# B&R Automation Studio project RobotNewEra (part 14)

#### HmiEditorLocal.typ - Local data types
```iecst
(********************************************************************
 * COPYRIGHT --
 ********************************************************************
 * Program: HmiEdit
 * File: HmiEdit.typ
 * Author: renj
 * Created: October 21, 2014
 ********************************************************************
 * Local data types of program HmiEdit
 ********************************************************************)

TYPE
	HmiEditorInternalStateType :
		(
		HMIEDITOR_WAIT,
		HMIEDITOR_READ,
		HMIEDITOR_LOADED,
		HMIEDITOR_WRITE_WAIT,
		HMIEDITOR_ERROR
		);
	HmiEditorInternalType : 	STRUCT
		State : HmiEditorInternalStateType;
	END_STRUCT;
END_TYPE
```

#### HmiEditorLocal.var - Local variables
```iecst
(********************************************************************
 * COPYRIGHT --
 ********************************************************************
 * Program: HmiEdit
 * File: HmiEdit.var
 * Author: renj
 * Created: October 21, 2014
 ********************************************************************
 * Local variables of program HmiEdit
 ********************************************************************)
VAR
	Internal : HmiEditorInternalType := (0);
	pSystem : REFERENCE TO System_Type;
	pCnc : REFERENCE TO Cnc_Type;
	pAxes : REFERENCE TO ARRAY[0..MAX_AX_MINUS_ONE] OF Axes_Type;
END_VAR
```

### Program Logical/HmiHandling/HmiEditor/HmiFileVar (IEC) - File Read Write

#### HmiFileCtrlVar.st - Implementation code
```iecst
(********************************************************************
 * COPYRIGHT --
 ********************************************************************
 * Program: HmiFile
 * File: HmiFileCtrlVar.st
 * Author: renj
 * Created: October 29, 2014
 ********************************************************************
 * Implementation of program HmiFile
 ********************************************************************)

PROGRAM _INIT

END_PROGRAM

PROGRAM _CYCLIC

	CASE Internal.State OF

		HMIFILE_IDLE:

			HmiFileCtrlVar.Output.Status.Busy := FALSE;

			IF HmiFileCtrlVar.Input.Command.Read THEN

				Internal.State := HMIFILE_OPEN;
				HmiFileCtrlVar.Output.Status.ReadOK := FALSE;
				HmiFileCtrlVar.Output.Status.Busy := TRUE;

			END_IF

			IF HmiFileCtrlVar.Input.Command.Write THEN

				Internal.State := HMIFILE_DELETE;
				HmiFileCtrlVar.Output.Status.WriteOK := FALSE;
				HmiFileCtrlVar.Output.Status.Busy := TRUE;
			END_IF

		HMIFILE_OPEN:

			FileOpen_0.enable	:= TRUE;
			FileOpen_0.pDevice 	:= ADR(HmiFileCtrlVar.Input.Parameter.FileDevice);
			FileOpen_0.pFile 	:= ADR(HmiFileCtrlVar.Input.Parameter.FileName);
			FileOpen_0.mode 	:= fiREAD_WRITE;
			(* FB Call *)
			FileOpen_0();

			(* Get FBK output information *)
			Internal.FileIdent := FileOpen_0.ident;
			wStatus := FileOpen_0.status;

			IF (wStatus = 0) THEN

				Internal.State := HMIFILE_READ;

			ELSIF (wStatus <> 65535) THEN
				(* Verify status (20708 -> File doesn't exist) *)
				IF (wStatus = 20708) THEN

				END_IF

				IF (wStatus = 20799) THEN
					wError := FileIoGetSysError();
				END_IF

				IF HmiFileCtrlVar.Input.Command.Read THEN

					HmiFileCtrlVar.Input.Command.Read := FALSE;

				ELSIF HmiFileCtrlVar.Input.Command.Write THEN

					HmiFileCtrlVar.Input.Command.Write := FALSE;

				END_IF

				Internal.State := HMIFILE_ERROR;

			END_IF

		HMIFILE_READ:

			(**** Read data from file ****)
			(* Initialize file read structure *)
			FileReadEx_0.enable		:= TRUE;
			FileReadEx_0.ident     	:= Internal.FileIdent;
			FileReadEx_0.pDest     	:= HmiFileCtrlVar.Input.Parameter.StringBufferAdr;
			FileReadEx_0.len	   	:= HmiFileCtrlVar.Input.Parameter.StringBufferSize;

			(* Call FBK *)
			FileReadEx_0();
			(* Get status *)
			wStatus := FileReadEx_0.status;
			(* Verify status *)
			IF wStatus = 0 THEN

				Internal.FileByte := FileReadEx_0.bytesread;

				Internal.State := HMIFILE_CLOSE;

			ELSIF (wStatus <> 65535) THEN

				IF (wStatus = 20799) THEN
					wError := FileIoGetSysError();
				END_IF

				IF HmiFileCtrlVar.Input.Command.Read THEN

					HmiFileCtrlVar.Input.Command.Read := FALSE;

				ELSIF HmiFileCtrlVar.Input.Command.Write THEN

					HmiFileCtrlVar.Input.Command.Write := FALSE;

				END_IF

				Internal.State := HMIFILE_ERROR;

			END_IF

		HMIFILE_DELETE:
			(* Initialize file delete structure *)
			FileDelete_0.enable  := 1;
			FileDelete_0.pDevice := ADR(HmiFileCtrlVar.Input.Parameter.FileDevice);
			FileDelete_0.pName   :=ADR(HmiFileCtrlVar.Input.Parameter.FileName);
			(* Call FBK *)
			FileDelete_0();
			(* Get status *)
			wStatus := FileDelete_0.status;

			(* Verify status *)
			IF wStatus = 0 THEN
				Internal.State := HMIFILE_CREATE;
			ELSIF (wStatus <> 65535) THEN

				IF (wStatus = 20799) THEN
					wError := FileIoGetSysError();
				END_IF

				IF HmiFileCtrlVar.Input.Command.Write THEN

					HmiFileCtrlVar.Input.Command.Write := FALSE;

				END_IF

				Internal.State := HMIFILE_ERROR;

			END_IF

		HMIFILE_CREATE:
			(* Initialize file create structure *)
			FileCreate_0.enable  := 1;
			FileCreate_0.pDevice := ADR(HmiFileCtrlVar.Input.Parameter.FileDevice);
			FileCreate_0.pFile   := ADR(HmiFileCtrlVar.Input.Parameter.FileName);
			(* Call FBK *)
			FileCreate_0();
			(* Get FBK output information *)
			Internal.FileIdent := FileCreate_0.ident;
			wStatus := FileCreate_0.status;
			(* Verify status *)
			IF wStatus = 0 THEN
				Internal.State := HMIFILE_WRITE;
			ELSIF (wStatus <> 65535) THEN

				IF (wStatus = 20799) THEN
					wError := FileIoGetSysError();
				END_IF

				IF HmiFileCtrlVar.Input.Command.Write THEN

					HmiFileCtrlVar.Input.Command.Write := FALSE;

				END_IF

				Internal.State := HMIFILE_ERROR;

			END_IF

		HMIFILE_WRITE:
			(**** WRITE File ****)
			(* Initialize file close structure *)
			FileWriteEx_0.enable	:= TRUE;
			FileWriteEx_0.ident		:= Internal.FileIdent;

			FileWriteEx_0.len		:= HmiFileCtrlVar.Input.Parameter.StringBufferSize;
			FileWriteEx_0.pSrc		:= HmiFileCtrlVar.Input.Parameter.StringBufferAdr;;

			(* Call FBK *)
			FileWriteEx_0();

			(* Get status *)
			wStatus := FileWriteEx_0.status;

			(* Verify status *)
			IF wStatus = 0 THEN
				Internal.State := HMIFILE_CLOSE;
			ELSIF (wStatus <> 65535) THEN

				IF (wStatus = 20799) THEN
					wError := FileIoGetSysError();
				END_IF

				IF HmiFileCtrlVar.Input.Command.Read THEN

					HmiFileCtrlVar.Input.Command.Read := FALSE;

				ELSIF HmiFileCtrlVar.Input.Command.Write THEN

					HmiFileCtrlVar.Input.Command.Write := FALSE;

				END_IF

				Internal.State := HMIFILE_ERROR;

			END_IF

		HMIFILE_CLOSE:
			(**** Close file ****)
			(* Initialize file close structure *)
			FileClose_0.enable	:= TRUE;
			FileClose_0.ident	:= Internal.FileIdent;

			(* Call FBK *)
			FileClose_0();

			(* Get status *)
			wStatus := FileClose_0.status;

			IF wStatus = 0 THEN

				IF HmiFileCtrlVar.Input.Command.Read THEN

					HmiFileCtrlVar.Output.Status.ReadOK := TRUE;

					HmiFileCtrlVar.Input.Command.Read := FALSE;

				ELSIF HmiFileCtrlVar.Input.Command.Write THEN

					HmiFileCtrlVar.Output.Status.WriteOK := TRUE;

					HmiFileCtrlVar.Input.Command.Write := FALSE;

				END_IF

				Internal.State := HMIFILE_IDLE;

			ELSIF (wStatus <> 65535) THEN

				IF (wStatus = 20799) THEN
					wError := FileIoGetSysError();
				END_IF

				IF HmiFileCtrlVar.Input.Command.Read THEN

					HmiFileCtrlVar.Input.Command.Read := FALSE;

				ELSIF HmiFileCtrlVar.Input.Command.Write THEN

					HmiFileCtrlVar.Input.Command.Write := FALSE;

				END_IF

				Internal.State := HMIFILE_ERROR;

			END_IF

		HMIFILE_ERROR:

			IF HmiFileCtrlVar.Input.Command.AckError THEN

				HmiFileCtrlVar.Input.Command.AckError := 0;
				Internal.State := HMIFILE_IDLE;

			END_IF

	END_CASE

END_PROGRAM
```

#### HmiFileVarLocal.var - Local variables
```iecst
(********************************************************************
 * COPYRIGHT --
 ********************************************************************
 * Program: HmiFile
 * File: HmiFileLocal.var
 * Author: renj
 * Created: October 29, 2014
 ********************************************************************
 * Local variables of program HmiFile
 ********************************************************************)
VAR
	FileOpen_0 : FileOpen := (0);
	FileClose_0 : FileClose := (0);
	FileReadEx_0 : FileReadEx := (0);
	FileDelete_0 : FileDelete := (0);
	FileCreate_0 : FileCreate := (0);
	FileWriteEx_0 : FileWriteEx := (0);
	wStatus : UINT := 0;
	wError : UINT := 0;
	Internal : HmiFileCtrlInternal_Type := (0);
END_VAR
```

### Package Logical/HmiHandling/HmiAlarm - Alarm Page

### Program Logical/HmiHandling/HmiAlarm/HmiAlarm (IEC) - Alarm Ctrl Page

#### HmiAlarm.st - Implementation code
```iecst
(********************************************************************
 * COPYRIGHT --
 ********************************************************************
 * Program: HmiAlarm
 * File: HmiAlarm.st
 * Author: renj
 * Created: October 14, 2014
 ********************************************************************
 * Implementation of program HmiAlarm
 ********************************************************************)

PROGRAM _INIT

END_PROGRAM

PROGRAM _CYCLIC

	IF HmiGlobal.PageControl.ActPage = PAGE_ALARM THEN
		IF (gUserLevel > 0) THEN

		END_IF
	ELSE

		RETURN;
	END_IF

END_PROGRAM
```

### Package Logical/HmiHandling/HmiJog - JogControl

### HmiJogGlobal.typ - Global data types
```iecst
(********************************************************************
 * COPYRIGHT --
 ********************************************************************
 * Package: HmiJog
 * File: HmiJogGlobal.typ
 * Author: renj
 * Created: January 06, 2015
 ********************************************************************
 * Data types of package HmiJog
 ********************************************************************)

TYPE
	HmiJogLayerDefaultType : 	STRUCT
		ButtoToolCheck : HmiButtonType;
		ButtonWorkObjectCheck : HmiButtonType;
		TextWorkObjectName : HmiTextType;
		TextToolName : HmiTextType;
		DropdownEulerQuan : HmiDropdownType;
		DropdownDegreeRad : HmiDropdownType;
		DropdownJointTCP : HmiDropdownType;
		NumericPos : ARRAY[0..6]OF HmiNumericType;
		NumericJogStep : HmiNumericType;
		TextPos : ARRAY[0..6]OF HmiTextType;
		TextPosUnit : ARRAY[0..5]OF HmiTextType;
		TextNotAvailable : HmiTextType;
		ButtonActSet : HmiButtonType;
		NumericPosSet : ARRAY[0..6]OF HmiNumericWithRangeType;
		TextActSet : HmiTextType;
		ButtonCheckVar : HmiButtonType;
		TextSetVar : HmiTextType;
		HotSpotFrameBrowse : HmiHotSpotType;
		HotSpotSetBrowse : HmiHotSpotType;
		HotSpotToolBrowse : HmiHotSpotType;
	END_STRUCT;
	HmiJogCtrlComponentsType : 	STRUCT
		LayerDefault : HmiJogLayerDefaultType;
	END_STRUCT;
	HmiJogCtrlType : 	STRUCT
		Components : HmiJogCtrlComponentsType;
	END_STRUCT;
END_TYPE
```

### HmiJogGlobal.var - Global variables
```iecst
(********************************************************************
 * COPYRIGHT --
 ********************************************************************
 * Package: HmiJog
 * File: HmiJogGlobal.var
 * Author: renj
 * Created: January 06, 2015
 ********************************************************************
 * Variables of package HmiJog
 ********************************************************************)
VAR
	HmiJog : HmiJogCtrlType := (0);
END_VAR
(*Global System Status*)
VAR
	JointAct : MXJointAxisType;
	PointAct : MXPointType := (0);
END_VAR
VAR RETAIN
	FrmSync : MXFrameType := (0);
	ToolSync : MXToolType;
	JointSync : MXAxisTargetType := (0);
	PointSync : MXPointType := (0);
	JointTCPSync : BOOL := FALSE;
END_VAR
VAR
	JointLimitsSync : ARRAY[0..5] OF HmiJointLimitType := [6(0)];
END_VAR
```

### Program Logical/HmiHandling/HmiJog/HmiJogCtrl (ANSIC) - Hmi Jog Ctrl

#### HmiJogCtrl.cpp - Implementation code
```cpp
/********************************************************************
 * COPYRIGHT --
 ********************************************************************
 * Program: HmiJogCtrl
 * File: HmiJogCtrl.cpp
 * Author: renj
 * Created: January 06, 2015
 ********************************************************************
 * Implementation of program HmiJogCtrl
 ********************************************************************/

#include <bur/plctypes.h>
#include <Arnc0mx.h>
#include <string>

#ifdef _DEFAULT_INCLUDES
#include <AsDefault.h>
#endif

unsigned long bur_heap_size = 0xFFFFF;

using namespace std;

#define PI 3.1415926535897932384626433832795028841971

void _INIT HmiJogCtrlInit(void)
{
	// Initialization
	HmiJog.Components.LayerDefault.NumericJogStep.Value = 2.0;
	for (int i = 0; i < 7; ++i)
		HmiJog.Components.LayerDefault.NumericPosSet[i].StatusDatapoint = 1;

	HmiJog.Components.LayerDefault.TextSetVar.StatusDatapoint = 1;
	HmiJog.Components.LayerDefault.ButtonCheckVar.StatusDatapoint = 1;

	JointSync.JointAxis[0] = JointSync.JointAxis[0];
	PointSync.Pos = PointSync.Pos;
	FrmSync.Pos = FrmSync.Pos;
	ToolSync.Frame = ToolSync.Frame;

}

void _CYCLIC HmiJogCtrlCyclic(void)
{

	string EditorFileName(HmiRetain.HmiEditor.Name);
	string EditorDevice(HmiRetain.HmiEditor.Device);

	string JogFileName(HmiRetain.HmiJog.Name);
	string JogDevice(HmiRetain.HmiJog.Device);

	if ((HmiGlobal.Address.CncAddress != 0) &&	(HmiGlobal.Address.SystemAddress != 0) && (HmiGlobal.Address.AxesAddress != 0))
	{
		pCnc = (Cnc_Type*) HmiGlobal.Address.CncAddress;
		pSystem = (System_Type*) HmiGlobal.Address.SystemAddress;
		pAxes = (Axes_Type (*)[13]) HmiGlobal.Address.AxesAddress;
	} else
	{
		return;
	}

	// If Robot not homed and Axis not homed and Actual Posiition shouldnt be shown("NOT AVAILABLE")
	if ((HmiRetain.HmiKeyControl.MechHomeOK && pSystem->Output.Status.HomingOk) || HmiJog.Components.LayerDefault.TextActSet.TextIndex == 1)
	{
		HmiJog.Components.LayerDefault.TextNotAvailable.StatusDatapoint = 1;
	}
	else
		HmiJog.Components.LayerDefault.TextNotAvailable.StatusDatapoint = 0;

	FrmSync = HmiRetain.HmiJog.Frame.Frame;
	ToolSync = HmiRetain.HmiJog.Tool.Tool;

	for (int i = 0; i < 6; ++ i)
	JointLimitsSync[i] = HmiRetain.HmiRobot.JointLimits[i];

	// Joint Act is Decoupled Position
	for (int i = 0; i < 6; ++ i)
		JointAct[i] = (*pAxes)[6+i].Output.Monitor.DecoupledPosition;

	// Calculate the TCP using the MXFunctions (Check if there are tools or Frames)
	if (ToolEnableSync)
		MXJointToPointEx((UDINT)&Robot_TRF, (double *)&JointAct, &Point, MX_CARDAN_XYZ_ANGLES, MX_TRF_TYPE_DIRECT, &ToolSync, &MX_FRAME_ZERO, &MX_POINT_ZERO);
	else
		MXJointToPointEx((UDINT)&Robot_TRF, (double *)&JointAct, &Point, MX_CARDAN_XYZ_ANGLES, MX_TRF_TYPE_DIRECT, &MX_TOOL_ZERO, &MX_FRAME_ZERO, &MX_POINT_ZERO);

	if (FrmEnableSync)
		MXToFrame(&FrmSync, &Point, &PointAct);
	else
		PointAct = Point;

	// Joint or TCP
	if (HmiJog.Components.LayerDefault.DropdownJointTCP.SelectedIndex == 0) // If Joint
	{
		// Do Once
		if (HmiJog.Components.LayerDefault.DropdownJointTCP.OldIndex == 1)
		{
			for (int i = 0; i < 6; ++i)
			{
				if (HmiJog.Components.LayerDefault.TextActSet.TextIndex == 1)
					HmiJog.Components.LayerDefault.NumericPosSet[i].Value = 0;
			}

		}

		for (int i = 0; i < 6; ++i)
		{
			HmiJog.Components.LayerDefault.TextPos[i].TextIndex = 0;
		}

		HmiJog.Components.LayerDefault.TextPos[6].StatusDatapoint = 1;
		HmiJog.Components.LayerDefault.NumericPos[6].StatusDatapoint = 1;
		HmiJog.Components.LayerDefault.NumericPosSet[6].StatusDatapoint = 1;

		if (HmiJog.Components.LayerDefault.DropdownDegreeRad.SelectedIndex == 0) // If Degree
		{
			// Do Once
			if (HmiJog.Components.LayerDefault.DropdownDegreeRad.OldIndex == 1)
			{
				for (int i = 0; i < 6; ++i)
				{
					if (HmiJog.Components.LayerDefault.TextActSet.TextIndex == 1)
						HmiJog.Components.LayerDefault.NumericPosSet[i].Value = 0;
				}
			}

			for (int i = 0; i < 6; ++i)
			{
				HmiJog.Components.LayerDefault.TextPosUnit[i].TextIndex = 2;
				HmiJog.Components.LayerDefault.NumericPosSet[i].Min = HmiRetain.HmiRobot.JointLimits[i].Min;
				HmiJog.Components.LayerDefault.NumericPosSet[i].Max = HmiRetain.HmiRobot.JointLimits[i].Max;
			}

			for (int i = 0; i < 6; ++i)
				HmiJog.Components.LayerDefault.NumericPos[i].Value = JointAct[i];

		} else //If Radian
		{
			// Do Once
			if (HmiJog.Components.LayerDefault.DropdownDegreeRad.OldIndex == 0)
			{

				if (HmiJog.Components.LayerDefault.TextActSet.TextIndex == 1)
				{
					for (int i = 0; i < 6; ++i)
						HmiJog.Components.LayerDefault.NumericPosSet[i].Value = 0;
				}
			}

			for (int i = 0; i < 6; ++i)
				{
				HmiJog.Components.LayerDefault.TextPosUnit[i].TextIndex = 3;
				HmiJog.Components.LayerDefault.NumericPosSet[i].Min = HmiRetain.HmiRobot.JointLimits[i].Min/180*PI;
				HmiJog.Components.LayerDefault.NumericPosSet[i].Max = HmiRetain.HmiRobot.JointLimits[i].Max/180*PI;
			}

			for (int i = 0; i < 6; ++i)
				HmiJog.Components.LayerDefault.NumericPos[i].Value = JointAct[i]/180 * PI;
		}

	} else // If TCP
	{
		// Do Once
		if (HmiJog.Components.LayerDefault.DropdownJointTCP.OldIndex == 0)
		{
			if (HmiJog.Components.LayerDefault.TextActSet.TextIndex == 1)
			{
				HmiJog.Components.LayerDefault.NumericPosSet[0].Value = HmiRetain.HmiRobot.HomePos.Pos.x;
				HmiJog.Components.LayerDefault.NumericPosSet[1].Value = HmiRetain.HmiRobot.HomePos.Pos.y;
				HmiJog.Components.LayerDefault.NumericPosSet[2].Value = HmiRetain.HmiRobot.HomePos.Pos.z;

				if (HmiJog.Components.LayerDefault.DropdownEulerQuan.SelectedIndex == 0)
				{
					for (int i = 0; i < 3; ++i)
						HmiJog.Components.LayerDefault.NumericPosSet[i + 3].Value = 0;
				} else
				{
					HmiJog.Components.LayerDefault.NumericPosSet[3].Value = 1;
					for (int i = 4; i < 7; ++i)
						HmiJog.Components.LayerDefault.NumericPosSet[i].Value = 0;
				}
			}

		}

		for (int i = 0; i < 3; ++i)
		{
			HmiJog.Components.LayerDefault.TextPos[i].TextIndex = 1;
			HmiJog.Components.LayerDefault.TextPosUnit[i].TextIndex = 1;
		}
		// Set the Limit for the Inputs
		HmiJog.Components.LayerDefault.NumericPosSet[0].Min = HmiRetain.HmiRobot.CartesianLimits[0].Min;
		HmiJog.Components.LayerDefault.NumericPosSet[1].Min = HmiRetain.HmiRobot.CartesianLimits[1].Min;
		HmiJog.Components.LayerDefault.NumericPosSet[2].Min = HmiRetain.HmiRobot.CartesianLimits[2].Min;

		HmiJog.Components.LayerDefault.NumericPosSet[0].Max = HmiRetain.HmiRobot.CartesianLimits[0].Max;
		HmiJog.Components.LayerDefault.NumericPosSet[1].Max = HmiRetain.HmiRobot.CartesianLimits[1].Max;
		HmiJog.Components.LayerDefault.NumericPosSet[2].Max = HmiRetain.HmiRobot.CartesianLimits[2].Max;

		HmiJog.Components.LayerDefault.NumericPos[0].Value = PointAct.Pos.x;
		HmiJog.Components.LayerDefault.NumericPos[1].Value = PointAct.Pos.y;
		HmiJog.Components.LayerDefault.NumericPos[2].Value = PointAct.Pos.z;

		if (HmiJog.Components.LayerDefault.DropdownEulerQuan.SelectedIndex == 0) // If Euler
		{
			// Do Once
			if (HmiJog.Components.LayerDefault.DropdownEulerQuan.OldIndex == 1)
			{
				for (int i = 3; i < 6; ++i)
				{
					if (HmiJog.Components.LayerDefault.TextActSet.TextIndex == 1)
						HmiJog.Components.LayerDefault.NumericPosSet[i].Value = 0;
				}
			}

			for (int i = 3; i < 6; ++i)
			{
				HmiJog.Components.LayerDefault.TextPos[i].TextIndex = 1;
			}

			HmiJog.Components.LayerDefault.TextPos[6].StatusDatapoint = 1;
			HmiJog.Components.LayerDefault.NumericPos[6].StatusDatapoint = 1;
			HmiJog.Components.LayerDefault.NumericPosSet[6].StatusDatapoint = 1;

			if (HmiJog.Components.LayerDefault.DropdownDegreeRad.SelectedIndex == 0) // If Degree
			{
				// Do Once
				if (HmiJog.Components.LayerDefault.DropdownDegreeRad.OldIndex == 1)
				{
					for (int i = 3; i < 6; ++i)
						{
						if (HmiJog.Components.LayerDefault.TextActSet.TextIndex == 1)
							HmiJog.Components.LayerDefault.NumericPosSet[i].Value = 0;
					}

				}

				for (int i = 3; i < 6; ++i)
					{
					HmiJog.Components.LayerDefault.TextPosUnit[i].TextIndex = 2;
					HmiJog.Components.LayerDefault.NumericPosSet[i].Min = -360;
					HmiJog.Components.LayerDefault.NumericPosSet[i].Max = 360;
				}

				for (int i = 3; i < 6; ++i)
					HmiJog.Components.LayerDefault.NumericPos[i].Value = PointAct.Orient.Angle[i - 3];

			} else // If Radian
			{
				// Do Once
				if (HmiJog.Components.LayerDefault.DropdownDegreeRad.OldIndex == 0)
				{
					for (int i = 3; i < 6; ++i)
						{

						if (HmiJog.Components.LayerDefault.TextActSet.TextIndex == 1)
							HmiJog.Components.LayerDefault.NumericPosSet[i].Value = 0;
					}
				}

				for (int i = 3; i < 6; ++i)
					{
					HmiJog.Components.LayerDefault.TextPosUnit[i].TextIndex = 3;
					HmiJog.Components.LayerDefault.NumericPosSet[i].Min = - 2 * PI;
					HmiJog.Components.LayerDefault.NumericPosSet[i].Max = 2 * PI;

					HmiJog.Components.LayerDefault.NumericPos[i].Value = PointAct.Orient.Angle[i - 3]/180*PI;
				}
			}

		} else // If Quanternion
		{
			// Do Once
			if (HmiJog.Components.LayerDefault.DropdownEulerQuan.OldIndex == 0)
			{
				if (HmiJog.Components.LayerDefault.TextActSet.TextIndex == 1)
				{
					HmiJog.Components.LayerDefault.NumericPosSet[3].Value = 1;
					for (int i = 4; i < 7; ++ i)
						HmiJog.Components.LayerDefault.NumericPosSet[i].Value = 0;
				}
			}

			HmiJog.Components.LayerDefault.TextPos[6].StatusDatapoint = 0;

			if (HmiJog.Components.LayerDefault.TextActSet.TextIndex == 0)
				HmiJog.Components.LayerDefault.NumericPos[6].StatusDatapoint = 0;
			else
				HmiJog.Components.LayerDefault.NumericPosSet[6].StatusDatapoint = 0;

			for (int i = 3; i < 6; ++i)
				{
				HmiJog.Components.LayerDefault.TextPos[i].TextIndex = 2;
				HmiJog.Components.LayerDefault.TextPosUnit[i].TextIndex = 0;
			}

			for (int i = 3; i < 7; ++i)
				{
				HmiJog.Components.LayerDefault.NumericPosSet[i].Min = -1;
				HmiJog.Components.LayerDefault.NumericPosSet[i].Max = 1;
			}

			LREAL RefAngle[3] = {0};
			MXConvertOrient(&PointAct.Orient, MX_QUATERNION, &Point.Orient, RefAngle); // Redo the Caculation for Quaternion
			PointAct.Orient = Point.Orient;

			for (int i = 3; i < 7; ++i)
				HmiJog.Components.LayerDefault.NumericPos[i].Value = PointAct.Orient.Angle[i - 3];

		}

	}

	// CNC Sync Variable For Jog Prog
	ToolEnableSync = HmiJog.Components.LayerDefault.ButtoToolCheck.Value == 1;
	FrmEnableSync = HmiJog.Components.LayerDefault.ButtonWorkObjectCheck.Value == 1;
	JogStepSync = HmiJog.Components.LayerDefault.NumericJogStep.Value;

	if (EditorFileName == "" || EditorDevice == "") // No Program/ Not Selected / Variable Name
	{
		HmiJog.Components.LayerDefault.TextToolName.TextIndex = 1; // No Prg
		HmiJog.Components.LayerDefault.TextWorkObjectName.TextIndex = 1; // No Prg
		HmiJog.Components.LayerDefault.ButtoToolCheck.Value = 0;
		HmiJog.Components.LayerDefault.ButtonWorkObjectCheck.Value = 0;
	} else
	{
		// Browse the Vars from the Editor Data Page
		if (HmiJog.Components.LayerDefault.HotSpotFrameBrowse.Value > HmiJog.Components.LayerDefault.HotSpotFrameBrowse.OldValue)
		{
			HmiGlobal.PageControl.SetPage = PAGE_EDITOR_DATA;
			HmiEditorCtrl.Components.PageData.LayerDefault.DropDownTypes.SelectedIndex = 2;
		}

		if (HmiJog.Components.LayerDefault.HotSpotToolBrowse.Value > HmiJog.Components.LayerDefault.HotSpotToolBrowse.OldValue)
		{
			HmiGlobal.PageControl.SetPage = PAGE_EDITOR_DATA;
			HmiEditorCtrl.Components.PageData.LayerDefault.DropDownTypes.SelectedIndex = 3;
		}

		if (JogFileName == "" || JogDevice == "")
		{
			HmiJog.Components.LayerDefault.TextToolName.TextIndex = 0; // Not Selected
			HmiJog.Components.LayerDefault.TextWorkObjectName.TextIndex = 0; // Not Selected
			HmiJog.Components.LayerDefault.ButtoToolCheck.Value = 0;
			HmiJog.Components.LayerDefault.ButtonWorkObjectCheck.Value = 0;
		} else
		{
			if (JogFileName != EditorFileName || JogDevice != EditorDevice)
			{
				HmiJog.Components.LayerDefault.TextToolName.TextIndex = 0; // Not Selected
				HmiJog.Components.LayerDefault.TextWorkObjectName.TextIndex = 0; // Not Selected
				HmiJog.Components.LayerDefault.ButtoToolCheck.Value = 0;
				HmiJog.Components.LayerDefault.ButtonWorkObjectCheck.Value = 0;
			} else
			{
				if (strcmp(HmiRetain.HmiJog.Tool.VarName, "") != 0)
					HmiJog.Components.LayerDefault.TextToolName.TextIndex = 2; // Tool
				else
					HmiJog.Components.LayerDefault.ButtoToolCheck.Value = 0;

				if (strcmp(HmiRetain.HmiJog.Frame.VarName, "") != 0)
					HmiJog.Components.LayerDefault.TextWorkObjectName.TextIndex = 2; // Frame
				else
					HmiJog.Components.LayerDefault.ButtonWorkObjectCheck.Value = 0;
			}
		}
	}

	// Set/Act Point for Jog to Certain Point/Joint
	if (HmiJog.Components.LayerDefault.ButtonActSet.Value > HmiJog.Components.LayerDefault.ButtonActSet.OldValue)
	{
		HmiJog.Components.LayerDefault.TextActSet.TextIndex = 1 - HmiJog.Components.LayerDefault.TextActSet.TextIndex;
		if (HmiJog.Components.LayerDefault.TextActSet.TextIndex == 0) // Act Position
		{
			for (int i = 0; i < 7; ++i)
			{
				HmiJog.Components.LayerDefault.NumericPosSet[i].StatusDatapoint = 1;
			}
			HmiJog.Components.LayerDefault.TextSetVar.StatusDatapoint = 1;
			HmiJog.Components.LayerDefault.ButtonCheckVar.StatusDatapoint = 1;

		} else // Set Position
		{

			HmiJog.Components.LayerDefault.TextSetVar.StatusDatapoint = 0;
			HmiJog.Components.LayerDefault.ButtonCheckVar.StatusDatapoint = 0;

			for (int i = 0; i < 7; ++i)
			{
				HmiJog.Components.LayerDefault.NumericPosSet[i].StatusDatapoint = 0;
			}

		}
	}

	if (HmiJog.Components.LayerDefault.TextActSet.TextIndex == 1) // Set Position Control
	{
		if (HmiJog.Components.LayerDefault.HotSpotSetBrowse.Value > HmiJog.Components.LayerDefault.HotSpotSetBrowse.OldValue &&
			(EditorFileName != "" && EditorDevice != ""))
		{
			HmiGlobal.PageControl.SetPage = PAGE_EDITOR_DATA;
			if (HmiJog.Components.LayerDefault.DropdownJointTCP.SelectedIndex == 0)
				HmiEditorCtrl.Components.PageData.LayerDefault.DropDownTypes.SelectedIndex = 1;
			else
				HmiEditorCtrl.Components.PageData.LayerDefault.DropDownTypes.SelectedIndex = 0;
		}

		if (EditorFileName == "" || EditorDevice == "")
		{
			HmiJog.Components.LayerDefault.ButtonCheckVar.Value = 0;
			HmiJog.Components.LayerDefault.TextSetVar.TextIndex = 1; // No Prg

		} else
		{
			if (JogFileName == "" || JogDevice == "")
			{
				HmiJog.Components.LayerDefault.ButtonCheckVar.Value = 0;
				HmiJog.Components.LayerDefault.TextSetVar.TextIndex = 0; // Not Selected
			} else
			{
				if (JogFileName != EditorFileName || JogDevice != EditorDevice)
				{
					HmiJog.Components.LayerDefault.ButtonCheckVar.Value = 0;
					HmiJog.Components.LayerDefault.TextSetVar.TextIndex = 0; // Not Selected
				} else
				{
					if (HmiRetain.HmiJog.Point.Set)
						HmiJog.Components.LayerDefault.TextSetVar.TextIndex = 2; // Point
					else if (HmiRetain.HmiJog.Joint.Set)
						HmiJog.Components.LayerDefault.TextSetVar.TextIndex = 3; // Joint
					else
					{
						HmiJog.Components.LayerDefault.TextSetVar.TextIndex = 0;
						HmiJog.Components.LayerDefault.ButtonCheckVar.Value = 0;
					}
				}
			}
		}

	}

	// Edge Detection
	HmiJog.Components.LayerDefault.ButtonActSet.OldValue = HmiJog.Components.LayerDefault.ButtonActSet.Value;
	HmiJog.Components.LayerDefault.HotSpotSetBrowse.OldValue = HmiJog.Components.LayerDefault.HotSpotSetBrowse.Value;
	HmiJog.Components.LayerDefault.HotSpotFrameBrowse.OldValue = HmiJog.Components.LayerDefault.HotSpotFrameBrowse.Value;
	HmiJog.Components.LayerDefault.HotSpotToolBrowse.OldValue = HmiJog.Components.LayerDefault.HotSpotToolBrowse.Value;
	HmiJog.Components.LayerDefault.DropdownDegreeRad.OldIndex = HmiJog.Components.LayerDefault.DropdownDegreeRad.SelectedIndex;
	HmiJog.Components.LayerDefault.DropdownEulerQuan.OldIndex = HmiJog.Components.LayerDefault.DropdownEulerQuan.SelectedIndex;
	HmiJog.Components.LayerDefault.DropdownJointTCP.OldIndex = HmiJog.Components.LayerDefault.DropdownJointTCP.SelectedIndex;

}
```

#### HmiJogLocal.var - Local variables
```iecst
(********************************************************************
 * COPYRIGHT --
 ********************************************************************
 * Program: HmiJogCtrl
 * File: HmiJogLocal.var
 * Author: renj
 * Created: January 06, 2015
 ********************************************************************
 * Local variables of program HmiJogCtrl
 ********************************************************************)
VAR
	pCnc : REFERENCE TO Cnc_Type;
	pSystem : REFERENCE TO System_Type;
	pAxes : REFERENCE TO ARRAY[0..MAX_AX_MINUS_ONE] OF Axes_Type;
	Point : MXPointType := (0);
	ToolEnableSync : BOOL := FALSE;
	FrmEnableSync : BOOL := FALSE;
	JogStepSync : LREAL := 0.0;
END_VAR
```

### Package Logical/ErrorHandling - Error Handling

### Error.typ
```iecst
(********************************************************************
 * COPYRIGHT -- Bernecker + Rainer
 ********************************************************************
 * Program: Error
 * File: Error.typ
 * Author: haged
 * Created: July 07, 2010
 ********************************************************************
 * Global data types of program Error
 ********************************************************************)

TYPE
	ErrorHandlingInputCommand_Type : 	STRUCT
		Acknowledge : BOOL;
		Reset : BOOL;
	END_STRUCT;
	ErrorHandlingInputPara_Type : 	STRUCT
		SystemAddress : UDINT;
		CncAddress : UDINT;
		AxesAddress : UDINT;
	END_STRUCT;
	ErrorHandlingInput_Type : 	STRUCT
		Parameter : ErrorHandlingInputPara_Type;
		Command : ErrorHandlingInputCommand_Type;
	END_STRUCT;
	ErrorHandlingOutputMon_Type : 	STRUCT
		ErrorHandlingAddress : UDINT;
		AlarmImage : ARRAY[0..MAX_ALARMS]OF BOOL;
	END_STRUCT;
	ErrorHandlingOutput_Type : 	STRUCT
		Monitor : ErrorHandlingOutputMon_Type;
		Status : ErrorHandlingStatus_Type;
	END_STRUCT;
	ErrorHandlingStatus_Type : 	STRUCT
		SystemError : BOOL;
		CncError : BOOL;
		Axeserror : BOOL;
	END_STRUCT;
	ErrorHandling_Type : 	STRUCT
		Input : ErrorHandlingInput_Type;
		Output : ErrorHandlingOutput_Type;
	END_STRUCT;
END_TYPE
```

### Program Logical/ErrorHandling/Error (IEC)

#### Error.st - Implementation code
```iecst
(********************************************************************
 * COPYRIGHT --  Bernecker + Rainer
 ********************************************************************
 * Program: Error
 * File: Error.st
 * Author: haged
 * Created: July 07, 2010
 ********************************************************************
 * Implementation of program Error
 ********************************************************************)

PROGRAM _INIT

	WarnMessage;

	Error.Output.Monitor.ErrorHandlingAddress := ADR(Error);
	RTInfo_0(enable := 1);
	cycT := RTInfo_0.cycle_time / 1000;

END_PROGRAM

PROGRAM _CYCLIC

	Error.Input.Parameter.AxesAddress := HmiGlobal.Address.AxesAddress;
	Error.Input.Parameter.CncAddress := HmiGlobal.Address.CncAddress;
	Error.Input.Parameter.SystemAddress := HmiGlobal.Address.SystemAddress;

	IF	(Error.Input.Parameter.AxesAddress <> 0)
		AND	(Error.Input.Parameter.CncAddress <> 0)
		AND	(Error.Input.Parameter.SystemAddress <> 0) THEN

		pAxes ACCESS Error.Input.Parameter.AxesAddress;
		pCnc ACCESS Error.Input.Parameter.CncAddress;
		pSystem ACCESS Error.Input.Parameter.SystemAddress;

	ELSE
		RETURN;
	END_IF

	WarnMessage[1] := NOT HmiRetain.HmiKeyControl.MechHomeOK;

	//Alarm monitor
	AlarmAcknDelay := AlarmAcknDelay + cycT;

	IF (AlarmAcknDelay > 500)THEN
		IF (pCnc[0].Output.State.Errorstop = 1) THEN
			IF (pCnc[0].Output.Error.Count = 0) THEN
				Error.Output.Monitor.AlarmImage[8] := 1;
			ELSE
				Error.Output.Monitor.AlarmImage[0] := 1;
			END_IF
		ELSE
			Error.Output.Monitor.AlarmImage[0] := 0;
			Error.Output.Monitor.AlarmImage[8] := 0;
		END_IF

		FOR i:= 6 TO MAX_AX_MINUS_ONE DO
			IF (pAxes[i].Output.State.Errorstop = 1)
				OR (pAxes[i].Output.Status.AxisError = 1)THEN
				IF (pAxes[i].Output.Error.Count = 0)  THEN
					Error.Output.Monitor.AlarmImage[i+3] := 1;
				ELSE
					Error.Output.Monitor.AlarmImage[i-5] := 1;
				END_IF
			ELSE
				Error.Output.Monitor.AlarmImage[i+3] := 0;
				Error.Output.Monitor.AlarmImage[i-5] := 0;
			END_IF
		END_FOR
	END_IF

	//HmiKeyControl.Output.Status.Error := 0;
	IF (HmiKeyControl.Output.Status.Error = 1) THEN

		IF (pCnc[0].Output.State.Moving = 1)THEN
			pCnc[0].Input.Command.Stop := 1;
		END_IF
	END_IF

	HmiKeyControl.Output.Status.Error := 0;

	FOR i:= 0 TO MAX_ALARMS DO					//axes alarm acknowledge
		IF (Error.Output.Monitor.AlarmImage[i] = 1) THEN
			HmiKeyControl.Output.Status.Error := 1;
			EXIT;
		END_IF
	END_FOR

	IF ((HmiKeyControl.Input.Command.StopKey <> 0) AND (OldStopKey = 0)
		AND (pSystem[0].Output.State.Errorstop = 0)) THEN
		Error.Input.Command.Acknowledge := 1;
	END_IF
	OldStopKey := HmiKeyControl.Input.Command.StopKey;

	IF (Error.Input.Command.Acknowledge = 1) THEN
		Error.Input.Command.Acknowledge := 0;
		pSystem[0].Input.Command.Acknowledge := 1;
		HmiKeyControl.Output.Status.Error := 0;
		FOR i:= 0 TO MAX_ALARMS DO					//axes alarm acknowledge
			Error.Output.Monitor.AlarmImage[i] := 0;
		END_FOR
		FOR i:= 0 TO WARN_MESSAGE_NUM DO
			WarnMessage[i]:=0;
		END_FOR
		AlarmAcknDelay := 0;

	END_IF

END_PROGRAM
```

#### ErrorPrv.var - Local variables
```iecst
(********************************************************************
 * COPYRIGHT --  Bernecker + Rainer
 ********************************************************************
 * Program: Error
 * File: ErrorPrv.var
 * Author: haged
 * Created: July 07, 2010
 ********************************************************************
 * Local variables of program Error
 ********************************************************************)
VAR
	pSystem : REFERENCE TO ARRAY[0..MAX_SYS_MINUS_ONE] OF System_Type;
	pCnc : REFERENCE TO ARRAY[0..MAX_CNC_MINUS_ONE] OF Cnc_Type; (*pTrf : REFERENCE TO ARRAY[0..MAX_CNC_MINUS_ONE] OF Trf_Type;*)
	pAxes : REFERENCE TO ARRAY[0..MAX_AX_MINUS_ONE] OF Axes_Type;
	Error : ErrorHandling_Type := (0);
	i : INT;
	cycT : DINT;
	RTInfo_0 : RTInfo;
	AlarmAcknDelay : UDINT;
	OldStopKey : BOOL;
END_VAR
```

### Package Logical/Recipe - Recipe Control

### RecipeGlobal.typ - Global data types
```iecst
(********************************************************************
 * COPYRIGHT --
 ********************************************************************
 * Package: Receipe
 * File: ReceipeGlobal.typ
 * Author: renj
 * Created: October 08, 2014
 ********************************************************************
 * Data types of package Receipe
 ********************************************************************)

TYPE
	RECIPE_DATA_USER_typ : 	STRUCT
		Reserve : USINT;
	END_STRUCT;
	RECIPE_DATA_SYSTEM_typ : 	STRUCT
		CurRcpIndex : UINT;
		RcpListName : ARRAY[0..LEN_RCP_NAME]OF STRING[NB_RECIPE];
		JointJogSpeed : REAL; (*deg/s*)
		PathJogSpeed : REAL; (*mm/s*)
		HomePosition : ARRAY[0..12]OF REAL;
		JogStepJoint : REAL;
		JogStepBase : REAL;
	END_STRUCT;
	RECIPE_DATA_typ : 	STRUCT
		System : RECIPE_DATA_SYSTEM_typ;
		User : RECIPE_DATA_USER_typ;
	END_STRUCT;
	RECIPE_COMMAND_typ : 	STRUCT
		Read : BOOL;
		UserDataWrite : BOOL;
		SysDataWrite : BOOL;
		Delete : BOOL;
		Rename : BOOL;
	END_STRUCT;
	RECIPE_MONITOR_typ : 	STRUCT
		CurrentRcpName : STRING[LEN_RCP_NAME];
		RcpInitOK : BOOL;
		ListRcpIndex : UINT;
		DataAddress : UDINT;
		RecipeAddress : UDINT;
	END_STRUCT;
	RECIPE_SET_PAR_typ : 	STRUCT
		NewRcpName : STRING[LEN_RCP_NAME];
	END_STRUCT;
	RECIPE_typ : 	STRUCT
		Cmd : RECIPE_COMMAND_typ;
		Monitor : RECIPE_MONITOR_typ;
		SetPar : RECIPE_SET_PAR_typ;
		Data : RECIPE_DATA_typ;
	END_STRUCT;
END_TYPE
```

### RecipeGlobal.var - Global variables
```iecst
(********************************************************************
 * COPYRIGHT --
 ********************************************************************
 * Package: Receipe
 * File: ReceipeGlobal.var
 * Author: renj
 * Created: October 08, 2014
 ********************************************************************
 * Variables of package Receipe
 ********************************************************************)
VAR CONSTANT
	NB_RECIPE : USINT := 20;
	LEN_RCP_NAME : USINT := 10;
	SG3 : USINT := 1;
	SG4 : USINT := 2;
	CPU_TYPE : USINT := SG4;
END_VAR
```

### Program Logical/Recipe/RecipeControl (ANSIC) - Recipe Control

#### RecipeControl.c - Implementation code
```c
/********************************************************************
 * COPYRIGHT --
 ********************************************************************
 * Program: ReceipeControl
 * File: ReceipeControl.c
 * Author: renj
 * Created: October 08, 2014
 ********************************************************************
 * Implementation of program ReceipeControl
 ********************************************************************/

#include <bur/plctypes.h>

#include <dataobj.h>
#include <string.h>           /*prototypes for asstring-library       */

#ifdef _DEFAULT_INCLUDES
	#include <AsDefault.h>
#endif

#if (CPU_TYPE == SG3)
_LOCAL DatObjMove_typ 		DOMove;
#endif

void _INIT ReceipeControlInit(void)
{
	if (Recipe.Data.System.CurRcpIndex >= NB_RECIPE)
		Recipe.Data.System.CurRcpIndex = NB_RECIPE-1;
	DataLen		= sizeof(Recipe.Data);
	SysDataLen	= sizeof(Recipe.Data.System);
	UserDataLen	= sizeof(Recipe.Data.User);
	RcpStep = 0;

	Recipe.Monitor.RecipeAddress = (UDINT)&Recipe;
	DOInfo.enable	= 1;
	DOInfo.pName	= (UDINT)"RecipeData";

	/* Call  FUB  */
	DatObjInfo(&DOInfo);

	/* Check the  status */
	if ((DOInfo.status == doERR_MODULNOTFOUND) || (DOInfo.status == doERR_ILLOBJTYPE)) /* Data module not found -> create a new one */
	{
		/* Initialize create structure */
		DOCreate.enable 	= 1;
		DOCreate.grp	 	= 0;
		DOCreate.pName 		= (UDINT)"RecipeData";		/*不能与任何任务名和其它数据模块名相同*/
		DOCreate.len 		= DataLen*NB_RECIPE;

#if (CPU_TYPE == SG3)
		DOCreate.MemType 	= doUSRRAM;
#elif (CPU_TYPE == SG4)
		DOCreate.MemType 	= doUSRROM;
#endif

		DOCreate.Option 	= 0;
		DOCreate.pCpyData 	= 0;

		/* Call FUB */
		DatObjCreate(&DOCreate);

		if (DOCreate.status == 0)
		{
#if (CPU_TYPE == SG3)
			/* Initialize move structure */
			DOMove.enable 	= 1;
			DOMove.ident 	= DOCreate.ident;
			DOMove.MemType 	= doFIXRAM;
			DOMove.Option 	= 0;
			/* Call FUB */
			DatObjMove(&DOMove);
			/* Verify status */
			if (DOMove.status == 0)
			{
				DoIdent = DOMove.identNew;
				strcpy(&ErrInfo[0],"DatObjMove executed correctly with no errors");
			}
			else
			{
				strcpy(&ErrInfo[0],"Error while moving data object(only SG3)");
			}

#elif (CPU_TYPE == SG4)	/* For SG4 targets */
			DoIdent = DOCreate.ident;
			strcpy(&ErrInfo[0],"DatObjCreate executed correctly with no errors");
#endif

		}
		else
		{
			strcpy(&ErrInfo[0],"Error while creating data object");
		}

#if	(CPU_TYPE == SG4)
		if (DOCreate.status == 0xFFFF)
		{
			strcpy(&ErrInfo[0],"DatObjCreate not yet complete - call FBK again (only SG4)");
		}
#endif
	}
	else
	{
		DoIdent = DOInfo.ident;
		strcpy(&ErrInfo[0],"DatObjInfo executed correctly with no errors");

		AdrOffset = 0;
		/* Initialize read structure */
		DORead.enable 		= 1;
		DORead.ident 		= DoIdent;
		DORead.Offset 		= AdrOffset;
		DORead.pDestination	= (UDINT)&Recipe.Data.System;
		DORead.len 			= SysDataLen;
		do
		{
			/* Call FUB */
			DatObjRead(&DORead);

			if (DORead.status == 0)
			{
				strcpy(&ErrInfo[0],"DatObjRead executed correctly with no errors");
				Recipe.Monitor.RcpInitOK = 1;
			}
			else if (DORead.status != 0xFFFF)
			{
				strcpy(&ErrInfo[0],"DatObjRead had executed with errors");
			}
		}
		while (DORead.status == 0xFFFF);

		AdrOffset = UserDataLen*Recipe.Data.System.CurRcpIndex + SysDataLen;
		/* Initialize read structure */
		DORead.enable 		= 1;
		DORead.ident 		= DoIdent;
		DORead.Offset 		= AdrOffset;
		DORead.pDestination	= (UDINT)&Recipe.Data.User;
		DORead.len 			= UserDataLen;

		do
		{
			/* Call FUB */
			DatObjRead(&DORead);

			if (DORead.status == 0)
			{
				strcpy(&ErrInfo[0],"DatObjRead executed correctly with no errors");
				strcpy(&Recipe.Monitor.CurrentRcpName[0],&Recipe.Data.System.RcpListName[Recipe.Data.System.CurRcpIndex][0]);
				Recipe.Monitor.RcpInitOK = 1;
			}
			else if (DORead.status != 0xFFFF)
			{
				strcpy(&ErrInfo[0],"DatObjRead had executed with errors");
			}
		}
		while (DORead.status == 0xFFFF);

	}/*end of if (DOInfo.status == doERR_MODULNOTFOUND)*/

	if (Recipe.Data.System.JointJogSpeed == 0)
		Recipe.Data.System.JointJogSpeed = 30;
	if (Recipe.Data.System.PathJogSpeed == 0)
		Recipe.Data.System.PathJogSpeed = 300;
	if (Recipe.Data.System.JogStepBase == 0)
		Recipe.Data.System.JogStepBase = 0.1;
	if (Recipe.Data.System.JogStepJoint == 0)
		Recipe.Data.System.JogStepJoint = 0.1;
}

void _CYCLIC ReceipeControlCyclic(void)
{
	switch(RcpStep)
	{
		case sIDLE:
			if ( Recipe.Cmd.Read )
			{
				RcpStep = sDAT_READ;
			}
			else if ( Recipe.Cmd.UserDataWrite )
			{
				RcpStep = sUSER_DAT_WRITE;
			}
			else if ( Recipe.Cmd.SysDataWrite )
			{
				RcpStep = sSYS_DAT_WRITE;
			}
			else if ( Recipe.Cmd.Rename )
			{
				strcpy(&Recipe.Data.System.RcpListName[Recipe.Monitor.ListRcpIndex][0],&Recipe.SetPar.NewRcpName[0]);
				Recipe.Cmd.Rename = 0;
				Recipe.Cmd.SysDataWrite = 1;
			}
			else if ( Recipe.Cmd.Delete )
			{
				strcpy(&Recipe.Data.System.RcpListName[Recipe.Monitor.ListRcpIndex][0],"");
				Recipe.Cmd.Delete = 0;
				Recipe.Cmd.SysDataWrite = 1;
			}
			break;

		case sDAT_READ:
			if (Recipe.Monitor.ListRcpIndex >= NB_RECIPE)
				Recipe.Monitor.ListRcpIndex = NB_RECIPE-1;

			AdrOffset = Recipe.Monitor.ListRcpIndex*UserDataLen + SysDataLen;

			/* Initialize read structure */
			DORead.enable 		= 1;
			DORead.ident 		= DoIdent;
			DORead.Offset 		= AdrOffset;
			DORead.pDestination	= (UDINT)&Recipe.Data.User;
			DORead.len 			= UserDataLen;

			/* Call FUB */
			DatObjRead(&DORead);

			if (DORead.status == 0)
			{
				strcpy(&ErrInfo[0],"DatObjRead executed correctly with no errors");
				Recipe.Cmd.Read = 0;
				strcpy(&Recipe.Monitor.CurrentRcpName[0],&Recipe.Data.System.RcpListName[Recipe.Monitor.ListRcpIndex][0]);
				Recipe.Data.System.CurRcpIndex = Recipe.Monitor.ListRcpIndex;
				Recipe.Cmd.SysDataWrite = 1;
				Recipe.Monitor.RcpInitOK = 1;
				RcpStep = sIDLE;
			}
			else if (DORead.status != 0xFFFF)
			{
				strcpy(&ErrInfo[0],"DatObjRead executed with errors");
				Recipe.Cmd.Read = 0;
				DORead.enable = 0;
				/* Call FUB */
				DatObjRead(&DORead);
				RcpStep = sIDLE;
			}
#if	(CPU_TYPE == SG4)
			if (DORead.status == 0xFFFF)
			{
				strcpy(&ErrInfo[0],"DatObjRead not yet complete - call FBK again (only SG4)");
			}
#endif
			break;

		case sUSER_DAT_WRITE:
			if (Recipe.Monitor.ListRcpIndex >= NB_RECIPE)
				Recipe.Monitor.ListRcpIndex = NB_RECIPE-1;

			AdrOffset = Recipe.Monitor.ListRcpIndex*UserDataLen + SysDataLen;

			/* Initialize read structure */
			DOWrite.enable 		= 1;
			DOWrite.ident 		= DoIdent;
			DOWrite.Offset 		= AdrOffset;
			DOWrite.pSource		= (UDINT)&Recipe.Data.User;
			DOWrite.len 		= UserDataLen;

			/* Call FUB */
			DatObjWrite(&DOWrite);

			if (DOWrite.status == 0)
			{
				strcpy(&ErrInfo[0],"UserDatObjWrite executed correctly with no errors");
				Recipe.Cmd.UserDataWrite = 0;
				strcpy(&Recipe.Monitor.CurrentRcpName[0],&Recipe.Data.System.RcpListName[Recipe.Monitor.ListRcpIndex][0]);
				Recipe.Data.System.CurRcpIndex = Recipe.Monitor.ListRcpIndex;
				Recipe.Cmd.SysDataWrite = 1;
				RcpStep = sIDLE;
			}
			else if (DOWrite.status != 0xFFFF)
			{
				strcpy(&ErrInfo[0],"UserDatObjWrite executed with errors");
				Recipe.Cmd.UserDataWrite = 0;
				DOWrite.enable = 0;
				/* Call FUB */
				DatObjWrite(&DOWrite);
				RcpStep = sIDLE;
			}
#if	(CPU_TYPE == SG4)
			if (DOWrite.status == 0xFFFF)
			{
				strcpy(&ErrInfo[0],"UserDatObjWrite not yet complete - call FBK again (only SG4)");
			}
#endif
			break;

		case sSYS_DAT_WRITE:
			AdrOffset = 0;

			/* Initialize read structure */
			DOWrite.enable 		= 1;
			DOWrite.ident 		= DoIdent;
			DOWrite.Offset 		= AdrOffset;
			DOWrite.pSource		= (UDINT)&Recipe.Data.System;
			DOWrite.len 		= SysDataLen;

			/* Call FUB */
			DatObjWrite(&DOWrite);

			if (DOWrite.status == 0)
			{
				strcpy(&ErrInfo[0],"SysDatObjWrite executed correctly with no errors");
				Recipe.Cmd.SysDataWrite = 0;
				RcpStep = sIDLE;
			}
			else if (DOWrite.status != 0xFFFF)
			{
				strcpy(&ErrInfo[0],"SysDatObjWrite executed with errors");
				Recipe.Cmd.SysDataWrite = 0;
				DOWrite.enable = 0;
				/* Call FUB */
				DatObjWrite(&DOWrite);
				RcpStep = sIDLE;
			}
#if	(CPU_TYPE == SG4)
			if (DOWrite.status == 0xFFFF)
			{
				strcpy(&ErrInfo[0],"SysDatObjWrite not yet complete - call FBK again (only SG4)");
			}
#endif
			break;

		default:
			RcpStep = sIDLE;
	}/*end of switch(RcpStep)*/
}
```

#### RecipeControlLocal.typ - Local data types
```iecst
(********************************************************************
 * COPYRIGHT --
 ********************************************************************
 * Program: ReceipeControl
 * File: ReceipeControlLocal.typ
 * Author: renj
 * Created: October 08, 2014
 ********************************************************************
 * Local data types of program ReceipeControl
 ********************************************************************)

TYPE
	RecipeState_Type :
		(
		sIDLE,
		sDAT_READ,
		sUSER_DAT_WRITE,
		sSYS_DAT_WRITE
		);
END_TYPE
```

#### RecipeControlLocal.var - Local variables
```iecst
(********************************************************************
 * COPYRIGHT --
 ********************************************************************
 * Program: ReceipeControl
 * File: ReceipeControlLocal.var
 * Author: renj
 * Created: October 08, 2014
 ********************************************************************
 * Local variables of program ReceipeControl
 ********************************************************************)
VAR
	Recipe : RECIPE_typ := (0);
	RcpStep : RecipeState_Type := sIDLE;
	DoIdent : UDINT := 0;
	DataLen : UDINT := 0;
	SysDataLen : UDINT := 0;
	UserDataLen : UDINT := 0;
	AdrOffset : UDINT := 0;
	ErrInfo : STRING[64] := '';
	DOCreate : DatObjCreate := (0);
	DOWrite : DatObjWrite := (0);
	DORead : DatObjRead := (0);
	DOInfo : DatObjInfo := (0);
END_VAR
```

### Package Logical/UserStd - User Management

### GlobalUserStd.var - Global variables
```iecst
(********************************************************************
 * COPYRIGHT --
 ********************************************************************
 * Package: UserStd
 * File: UserStd.var
 * Author: Liub
 * Created: January 16, 2012
 ********************************************************************
 * Variables of package UserStd
 ********************************************************************)
VAR
	gUserLevel : USINT := 0;
END_VAR
```

### Program Logical/UserStd/UserStd (ANSIC) - 用户管理

#### UserStd.c - Implementation code
```c
/********************************************************************
 * COPYRIGHT --
 ********************************************************************
 * Program: User
 * File: User.c
 * Author: Liub
 * Created: January 16, 2012
 ********************************************************************
 * Implementation of program User
 ********************************************************************/
/*任务功能*/
/*日期时间设定 用户登录推出 密码级别管理*/
/* Level 1 - machine worker 机长*/
/* Level 2 - factory worker 班长*/
/* Level 3 - 设备管理员 */
/* Level 4 - 厂方人员*/
#include <bur/plctypes.h>
#include <string.h>
#ifdef _DEFAULT_INCLUDES
	#include <AsDefault.h>
#endif

/*step for task*/
#define		STEP_WAIT_COMMAND			0
#define		STEP_LOG_IN			        100
#define		STEP_LOG_OUT_TO_PRE			200
#define		STEP_LOG_OUT			    300
#define		STEP_NEW_USER				400
#define		STEP_DEL_USER				500
#define		STEP_SAVE_DATAOBJ           550
#define		STEP_REFRESH_VIS            600
/*info to vis*/
#define		MAX_NO_INFO				    15
#define		INFO_CREATE_OK			    1
#define		INFO_LOAD_OK			    2
#define		INFO_WRITE_OK			    3
#define		INFO_DEL_OK				    4
#define		INFO_HAVE_NAME			    5		/*have name can not save at here*/
/*alarm to vis*/
#define		ERR_CREATE_MODULE		    16		/*Alarm*/
#define		ERR_LOAD				    17
#define		ERR_WRITE				    18
#define		ERR_DEL					    19
#define		ERR_REFRESH_NAME            20
#define		ERR_STRU_NAME               21      /*data object structure name can not find*/
#define		ERR_DATA_OBJ_SIZE           22      /*data object size has changed,delete old one restart again*/
#define		ERR_MEM_ALLOC               23      /*memalloc error*/

void _INIT UserINIT(void)
{
	/* TODO: Add code here */
    /*constant variable declear,otherwise buile warning happen*/
    constant = MAX_PASSWORD_LENGTH;
    constant = MAX_USER_MINUS_ONE;
    constant = MAX_USER_NAME_LENGTH;
    /*Get data object info*/
    dataObjInfo.enable = 1;
    dataObjInfo.pName = (UDINT)PASSWORD_DATA_NAME;
    DatObjInfo(&dataObjInfo);
    if(dataObjInfo.status == 0)                           /*数据模块存在    --  获取id*/
    {
        ident = dataObjInfo.ident;
        dataObjSize = dataObjInfo.len;
        /**********Read*********/
        dataObjRead.enable 		= 1;
        dataObjRead.ident 		= ident;
        dataObjRead.Offset 		= 0;
        dataObjRead.pDestination	= (UDINT) &userData;
        dataObjRead.len 			= sizeof (userData);

        /* Call FUB */
        DatObjRead(&dataObjRead);
        if(dataObjRead.status==0)
        {
        }
        else if(dataObjRead.status!=65535)
        {
            errorInfo = ERR_LOAD;		/*Datamodule read error Please restart again*/
            errorNumber = dataObjRead.status;
        }
    }
    else if(dataObjInfo.status == doERR_MODULNOTFOUND)    /*数据模块不存在   --  创建数据模块*/
    {
        dataObjSize             = sizeof (userData_typ);
        dataObjCreate.enable    = 1;
        dataObjCreate.grp	    = 0;
        dataObjCreate.pName     = (UDINT)PASSWORD_DATA_NAME;
        dataObjCreate.len	    = sizeof (userData);
        dataObjCreate.MemType   = 2;		/*doUSRROM  2 */
        dataObjCreate.Option	= 0;		/*with  checksum*/
        dataObjCreate.pCpyData  = 0;
        DatObjCreate(&dataObjCreate);
        if(dataObjCreate.status == 0)
        {
            ident = dataObjCreate.ident;
        }
        else
        {
            errorInfo = ERR_CREATE_MODULE;		/*Datamodule create error Please restart again*/
            errorNumber = dataObjCreate.status;
        }
    }
    /*data object size maybe a little bigger(1-3) than structure size because of offset*/
    /*data structure size must smaller than data object size*/
    dataStruSize = sizeof (userData);
    userData.level[0] = userData.level[0];
    /*dataObjSize is multiple of 4,so some time it is a little bigger than dataStruSize*/
    /*for example dataStruSize=3,dataObjSize=4*/
    if((dataObjSize - dataStruSize)>=4 || (dataStruSize > dataObjSize))
    {
        errorInfo = ERR_DATA_OBJ_SIZE;
        initError = 1;
    }
}

void _CYCLIC UserCYCLIC(void)
{
    /* TODO: Add code here */
    if(initError == 1) return;
    /*Only high password level can quit to low password level*/
    if((curUser.level > preUser.level) && (preUser.userName[0] != 0))
    {
        disableLogOutToPre = 0;		/*Show this button*/
    }
    else
    {
        disableLogOutToPre = 1;		/*do not show button on vis*/
    }
    switch(userStep)
    {
        case STEP_WAIT_COMMAND:
            if(cmdLogIn)
            {
                cmdLogIn = 0;
                if(curPassword[0] != 0)	/*password not empty*/
                {
                    userStep = STEP_LOG_IN;
                }
            }
            else if(cmdLogOutToPre)
            {
                cmdLogOutToPre = 0;
                userStep = STEP_LOG_OUT_TO_PRE;
            }
            else if(cmdLogOut)
            {
                cmdLogOut = 0;
                userStep = STEP_LOG_OUT;
            }
            else if(cmdNewUser)
            {
                cmdNewUser = 0;
                if(newUser.userName[0] != 0)
                {
                    userStep = STEP_NEW_USER;
                }
            }
            else if(cmdDelUser)
            {
                cmdDelUser = 0;
                if(visUserData.userName[focusIndex][0] != 0)
                {
                    userStep = STEP_DEL_USER;
                }
            }
            break;
        case STEP_LOG_IN:
            if(strcmp(curPassword,USER_ADMIN_PASSWORD)==0 )     /*system administrator password---3652101002101905469--091321186290913--*/
            {
                memcpy(&preUser,&curUser,sizeof(curUser));
                curUser.level = 4;
                strcpy(curUser.userName,"admin");
                userStep = STEP_REFRESH_VIS;
                curPassword[0] = 0;	                            /*Clear password*/
                break;
            }

            for(i=0;i<MAX_USER;i++)
            {
                result = strcmp(curPassword,userData.password[i]);
                if(result == 0)			/*Found a same password*/
                {
                    /*Transfer data to preUser*/
                    memcpy(&preUser,&curUser,sizeof(curUser));
                    /*Get curUser data*/
                    strcpy(curUser.userName,userData.userName[i]);
                    strcpy(curUser.password,userData.password[i]);
                    curUser.level = userData.level[i];

                    userStep = STEP_REFRESH_VIS;
                    curPassword[0] = 0;	/*Clear password*/
                    break;
                }
            }
            if(i == MAX_USER)
            {
                userStep = STEP_WAIT_COMMAND;
            }
            curPassword[0] = 0;	                /*Clear password*/
            memset(&newUser,0,sizeof(newUser));	/*clear new user data*/
            break;
        case STEP_LOG_OUT_TO_PRE:
            memcpy(&curUser,&preUser,sizeof(curUser));
            memset(&newUser,0,sizeof(newUser));	/*clear new user data*/
            userStep = STEP_REFRESH_VIS;
            break;
        case STEP_LOG_OUT:
            memset(&curUser,0,sizeof(curUser));
            memset(&preUser,0,sizeof(preUser));
            memset(&newUser,0,sizeof(newUser));	/*clear new user data*/
            userStep = STEP_REFRESH_VIS;
            break;
        case STEP_NEW_USER:
            if(newUser.password[0] == 0)
            {
                userStep = STEP_WAIT_COMMAND;
            }
            else
            {
                /*Save user to dataobj*/
                for(i=0;i<MAX_USER;i++)
                {
                    if(userData.userName[i][0] == 0)/*this is empty*/
                    {
                        strcpy(userData.userName[i],newUser.userName);
                        strcpy(userData.password[i],newUser.password);
                        if(newUser.level == 0)              newUser.level = 1;		        /*limit user level*/
                        if(newUser.level > MAX_USER_LEVEL)  newUser.level = MAX_USER_LEVEL; /*limit user level*/
                        userData.level[i] = newUser.level;
                        /*clear new user info*/
                        newUser.userName[0] = 0;
                        newUser.password[0] = 0;
                        newUser.level       = 0;

                        userStep = STEP_SAVE_DATAOBJ;
                        break;
                    }
                }
                if(i == MAX_USER)
                {
                    userStep = STEP_WAIT_COMMAND;
                }
            }
            break;
        case STEP_DEL_USER:
            if(visUserData.userName[focusIndex][0] != 0)	/*Choose is not empty*/
            {
                memset(&userData.userName[visUserIndex[focusIndex]],0,sizeof(userData.userName[0]));
                memset(&userData.password[visUserIndex[focusIndex]],0,sizeof(userData.password[0]));
                userData.level[visUserIndex[focusIndex]] = 0;
                userStep = STEP_SAVE_DATAOBJ;
            }
            break;
        case STEP_SAVE_DATAOBJ:
            dataObjWrite.enable 	= 1;
            dataObjWrite.ident 	= ident;
            dataObjWrite.Offset 	= 0;
            dataObjWrite.pSource = (UDINT) &userData;
            dataObjWrite.len 	= sizeof (userData);

            /* Call FUB */
            DatObjWrite(&dataObjWrite);
            if(dataObjWrite.status==0)
            {
                userStep = STEP_REFRESH_VIS;
            }
            else if(dataObjWrite.status!=65535)
            {
                userStep = STEP_WAIT_COMMAND;
            }
            break;
        case STEP_REFRESH_VIS:	/*user can only see level lower than himself*/
            memset(&visUserData,0,sizeof(visUserData));
            k = 0;
			// Added by RJ 2014/12/29
			HmiKeyControl.Components.LayerLogin.Layer.StatusDatapoint = 1;
            if(curUser.level != 0)
            {
                for(i=0;i<curUser.level;i++)
                {
                    for(j=0;j<MAX_USER;j++)
                    {
                        if(userData.level[j]==(i+1))
                        {
                            strcpy(visUserData.userName[k],userData.userName[j]);
                            strcpy(visUserData.password[k],userData.password[j]);
                            visUserData.level[k] = userData.level[j];
                            visUserIndex[k] = j;
                            k++;
                        }
                    }
                }
            }
            userStep = STEP_WAIT_COMMAND;
            break;
    }
    gUserLevel = curUser.level;
}
```

#### User.typ - Local data types
```iecst
(********************************************************************
 * COPYRIGHT --
 ********************************************************************
 * Program: User
 * File: User.typ
 * Author: Liub
 * Created: January 16, 2012
 ********************************************************************
 * Local data types of program User
 ********************************************************************)

TYPE
	userData_typ : 	STRUCT  (*Save to data object*)
		userName : ARRAY[0..MAX_USER_MINUS_ONE]OF STRING[MAX_USER_NAME_LENGTH];
		password : ARRAY[0..MAX_USER_MINUS_ONE]OF STRING[MAX_PASSWORD_LENGTH];
		level : ARRAY[0..MAX_USER_MINUS_ONE]OF USINT;
	END_STRUCT;
	user_typ : 	STRUCT  (*user interface*)
		userName : STRING[MAX_USER_NAME_LENGTH];
		password : STRING[MAX_PASSWORD_LENGTH];
		level : USINT;
	END_STRUCT;
END_TYPE
```

#### User.var - Local variables
```iecst
(********************************************************************
 * COPYRIGHT --
 ********************************************************************
 * Program: User
 * File: User.var
 * Author: Liub
 * Created: January 16, 2012
 ********************************************************************
 * Local variables of program User
 ********************************************************************)
(*-----------------------------------------------------------------------*)
(*以下常量可以按照需求修改，建议不要修改*)
(*-----------------------------------------------------------------------*)
VAR CONSTANT
	MAX_USER : USINT := 8; (*修改此常量数值会改变数据模块大小，需要删除已创建的数据模块*)
	MAX_USER_MINUS_ONE : USINT := MAX_USER-1; (*请勿修改*)
	MAX_USER_NAME_LENGTH : USINT := 8; (*修改此常量数值会改变数据模块大小，需要删除已创建的数据模块*)
	MAX_PASSWORD_LENGTH : USINT := 8; (*修改此常量数值会改变数据模块大小，需要删除已创建的数据模块*)
	USER_ADMIN_PASSWORD : STRING[MAX_PASSWORD_LENGTH] := '123'; (*管理员密码*)
	PASSWORD_DATA_NAME : STRING[10] := 'myUser'; (*创建数据模块名称*)
END_VAR
(*-----------------------------------------------------------------------*)
(*以下常量请勿修改*)
(*-----------------------------------------------------------------------*)
VAR CONSTANT
	MAX_USER_LEVEL : USINT := 4; (*最高密码等级*)
END_VAR
(*-----------------------------------------------------------------------*)
(*命令接口*)
(*-----------------------------------------------------------------------*)
VAR
	cmdLogIn : USINT := 0;
	cmdLogOutToPre : USINT := 0;
	cmdLogOut : USINT;
	cmdNewUser : USINT := 0;
	cmdDelUser : USINT := 0;
END_VAR
(*Interface to Visu*)
VAR
	userData : userData_typ := (0); (*Save to data object*)
	visUserIndex : ARRAY[0..MAX_USER_MINUS_ONE] OF USINT := [10(0)];
	visUserData : userData_typ := (0); (*Show to vis,can be change by different password level*)
	preUser : user_typ := (0);
	curUser : user_typ := (0);
	newUser : user_typ := (0);
	focusIndex : UINT := 0;
	curPassword : STRING[10];
END_VAR
(*Variable Output*)
VAR
	errorInfo : UINT := 0;
	errorNumber : UINT := 0;
	disableLogOutToPre : UINT := 0; (*output: status of button logOutToPre*)
END_VAR
(*-----------------------------------------------------------------------*)
(*The following is internal variable do not need modify *)
(*-----------------------------------------------------------------------*)
(*data object structure*)
VAR
	dataObjCreate : DatObjCreate := (0);
	dataObjInfo : DatObjInfo := (0);
	dataObjWrite : DatObjWrite := (0);
	dataObjRead : DatObjRead := (0);
END_VAR
(*Other*)
VAR
	dataStruSize : UINT := 0;
	dataObjSize : UINT := 0;
	initError : USINT := 0;
	ident : UDINT := 0;
	userStep : UINT := 0;
	result : UINT := 0;
	k : USINT := 0;
	j : USINT := 0;
	i : USINT := 0;
	constant : DINT := 0;
END_VAR
```

- Visualisation Logical/Visualization (not shown)

### Data object Logical/GmcIpConfig/gmcipcbr (Cnc, version 2.48.1)

- gmcipcbr.cnc (not shown)

### Data object Logical/GmcIpConfig/gmcipcfg (Cnc, version 2.48.1)

#### gmcipcfg.cnc
```
CONFIG:
  LANG_INCLUDE gmcipmxd (LangName=IEC-ST, DataObject=Yes, IfNotExist=Error, Scope=NC_GLOBAL, RequireFnIgnore=MXConvertOrient)
  XML_INCLUDE gmcipvar (IfNotExist=Warn)
  XML_INCLUDE gmcipfun (IfNotExist=Warn)
  XML_INCLUDE gmcipfub (IfNotExist=Warn)
  MPQUEUE (NumPackets=200, LookaheadMinBlocks=5, LookaheadMaxBlocks=20, LookaheadMode=any, MaxPathJobs=256)
  MONITOR (MaxPathStackEvents=1024)
  MPLOG (MaxBuffers=10, MinBuffers=4, EarlyCircleBufferLookahead=2, DefaultBufferSize=131072, TaskCycleDelay=1, FileDevice=mplog*, MaxLogFiles=20, MaxLogFileSize=1048576, CopyLineTextMaxChars=80)
  AXES (StandardCNCAxes=Yes)
  FUBOutputs:
    FUBOutput PLCOpen:
      ERROR (condition=$Error == 1)
      BUSY (condition=$Busy == 1)
    FUBOutput BuR:
      ERROR (condition=$status != 65535 && $status != 0)
      BUSY (condition=$status == 65535)
  FUNCTIONS:
    FUNC LEN (DeclareName=__LEN, AlwaysDeclare=Yes, RetType=INT)
      ARG IN (Type=STRING)
    FUNC LEFT (DeclareName=__LEFT, AlwaysDeclare=Yes, RetType=STRING, RetRef=Yes)
      ARG IN (Type=STRING)
      ARG L (Type=INT)
    FUNC RIGHT (DeclareName=__RIGHT, AlwaysDeclare=Yes, RetType=STRING, RetRef=Yes)
      ARG IN (Type=STRING)
      ARG L (Type=INT)
    FUNC MID (DeclareName=__MID, AlwaysDeclare=Yes, RetType=STRING, RetRef=Yes)
      ARG IN (Type=STRING)
      ARG L (Type=INT)
      ARG P (Type=INT)
    FUNC CONCAT (DeclareName=__CONCAT, AlwaysDeclare=Yes, RetType=STRING, RetRef=Yes)
      ARG IN1 (Type=STRING)
      ARG IN2 (Type=STRING)
    FUNC INSERT (DeclareName=__INSERT, AlwaysDeclare=Yes, RetType=STRING, RetRef=Yes)
      ARG IN1 (Type=STRING)
      ARG IN2 (Type=STRING)
      ARG P (Type=INT)
    FUNC DELETE (DeclareName=__DELETE, AlwaysDeclare=Yes, RetType=STRING, RetRef=Yes)
      ARG IN (Type=STRING)
      ARG L (Type=INT)
      ARG P (Type=INT)
    FUNC REPLACE (DeclareName=__REPLACE, AlwaysDeclare=Yes, RetType=STRING, RetRef=Yes)
      ARG IN1 (Type=STRING)
      ARG IN2 (Type=STRING)
      ARG L (Type=INT)
      ARG P (Type=INT)
    FUNC FIND (DeclareName=__FIND, AlwaysDeclare=Yes, RetType=INT)
      ARG IN1 (Type=STRING)
      ARG IN2 (Type=STRING)
  XML_INCLUDE gmcipuc (IfNotExist=Warn)
```

### Data object Logical/GmcIpConfig/gmcipcsm (Cnc, version 2.48.1)

#### gmcipcsm.cnc
```
Root (LangModule=ailgcode, Version=1.0)
  Constants:
    NumAxes = 15 (Type=INT)
  Preprocess:
    PP_RULE_STOPRE (Search=STOPRE, Replace=G172)
    PP_RULE_CIP (Search=CIP:\W, Replace=G102, IsPattern=Yes)
  Types:
    RotationAngleSpecifier (type=ENUM, EnumType=REGEXP, Value6=H)
    RadiusSpecifier (type=ENUM, EnumType=REGEXP, Value1=R\s*=, Value2=CR\s*=)
    InterpolParam (type=ENUM, EnumType=REGEXP, Value0=I, Value1=J, Value2=K, Value100=G161\s*I, Value101=G161\s*J, Value102=G161\s*K, Value200=G162\s*I, Value201=G162\s*J, Value202=G162\s*K, Value0300=I\s*=\s*AC, Value0301=J\s*=\s*AC, Value0302=K\s*=\s*AC, Value0400=I\s*=\s*IC, Value0401=J\s*=\s*IC, Value0402=K\s*=\s*IC)
    CirclePointParam (type=ENUM, EnumType=REGEXP, Value0=I1\s*=, Value1=J1\s*=, Value2=K1\s*=, Value100=G161\s*I1\s*=, Value101=G161\s*J1\s*=, Value102=G161\s*K1\s*=, Value200=G162\s*I1\s*=, Value201=G162\s*J1\s*=, Value202=G162\s*K1\s*=, Value0300=I1\s*=\s*AC, Value0301=J1\s*=\s*AC, Value0302=K1\s*=\s*AC, Value0400=I1\s*=\s*IC, Value0401=J1\s*=\s*IC, Value0402=K1\s*=\s*IC)
    RPYAngleName (type=ENUM, EnumType=REGEXP, Value1=ROLL, Value0=PITCH, Value2=YAW)
    EulerAngleName (type=ENUM, EnumType=REGEXP, Value3=PHI, Value4=THETA, Value5=PSI)
    RotaryVectorName (type=ENUM, EnumType=REGEXP, Value0=P\s*=, Value1=Q\s*=, Value2=R\s*=)
    DwellTime (type=FLOAT)
    RParamIndex (type=INT, MinValue=0, MaxValue=999)
    EXParamIndex (type=INT, MinValue=0, MaxValue=99)
    MParamIndex (type=INT, MinValue=0, MaxValue=99)
    Byte (type=INT, MinValue=0, MaxValue=255)
    Word (type=INT, MinValue=-32768, MaxValue=32767)
    Long (type=INT)
    AxisAccelPercentage (type=FLOAT, MinValue=0.0000001, MaxValue=100)
  PVMacros:
    SAVE (ArrayDims=0, Group=500)
      CALL = Info(:id:52101, msg:"Save Modal GCode State NOT SUPPORTED YET":);
  SysVars:
    P_F $P_F:
      GET = return @%_CNC.v_ncprog;
    P_GG $P_GG:
      GET = return @%_CNC.typ_ncblock;
    LIM_PATH_V $LIM_PATH_V:
      GET = return %_CNC.lim_path_v;
      SET:
        ARG (ref=EXPR, DataType=FLOAT)
    LIM_PATH_ACC_P $LIM_PATH_ACC_P:
      GET = return %_CNC.lim_path_acc_p;
      SET:
        ARG (ref=EXPR, DataType=FLOAT)
    LIM_PATH_ACC_N $LIM_PATH_ACC_N:
      GET = return %_CNC.lim_path_acc_n;
      SET:
        ARG (ref=EXPR, DataType=FLOAT)
    S_JUMP_T $S_JUMP_T:
      GET = return %_CNC.s_jump_t;
      SET:
        ARG (ref=EXPR, DataType=FLOAT)
    RADIUS_ERR $RADIUS_ERR:
      GET = return %_CNC.radius_err;
      SET:
        ARG (ref=EXPR, DataType=FLOAT)
    V_JUMP_T $V_JUMP_T:
      GET = return %_CNC.v_jump_t;
      SET:
        ARG (ref=EXPR, DataType=FLOAT)
    LIM_AX_ACC $LIM_AX_ACC (ArrayDims=1)
      GET = return %_AX.a_max_ncdy[$[1]];
      SET:
        ARG (ref=EXPR, DataType=FLOAT)
    LIM_ACC ACC (ArrayDims=1)
      GET = return %_AX.a_max_ncdy[$[1]] / %_AX.a_max[$[1]] * 100.0;
      SET:
        ARG (ref=EXPR, DataType=AxisAccelPercentage)
    LIM_AX_V $LIM_AX_V (ArrayDims=1)
      GET = return %_AX.v_max_ncdy[$[1]];
      SET:
        ARG (ref=EXPR, DataType=FLOAT)
    AX_A_JUMP $AX_A_JUMP (ArrayDims=1)
      GET = return %_AX.a_jump_ncdy[$[1]];
      SET:
        ARG (ref=EXPR, DataType=FLOAT)
    AX_V_JUMP $AX_V_JUMP (ArrayDims=1)
      GET = return %_AX.v_jump_ncdy[$[1]];
      SET:
        ARG (ref=EXPR, DataType=FLOAT)
    AX_T_INPOS $AX_T_INPOS (ArrayDims=1)
      GET = return %_AX.t_inpos[$[1]];
    AX_T_IN_POS $AX_T_IN_POS (ArrayDims=1)
      GET = return %_AX.t_inpos[$[1]];
    AX_T_JOLT $AX_T_JOLT (ArrayDims=1)
      GET = return %_AX.t_jolt_ax[$[1]];
    PATH_T_JOLT $PATH_T_JOLT:
      GET = return %_CNC.path_t_jolt;
    LIM_PATH_ACC_P_INI $LIM_PATH_ACC_P_INI:
      GET = return %_CNC.lim_path_acc_p_ini;
    LIM_PATH_ACC_N_INI $LIM_PATH_ACC_N_INI:
      GET = return %_CNC.lim_path_acc_n_ini;
    AA_IM $AA_IM (ArrayDims=1)
      GET = return @%_AX.set_pos_mcs[$[1]];
    AA_IW $AA_IW (ArrayDims=1)
      GET = return @%_AX.set_pos[$[1]];
    P_SIM $P_SIM (ArrayDims=1)
      GET = return %_AX.sim_status[$[1]];
    MA_MAX_AX_ACCEL $MA_MAX_AX_ACCEL (ArrayDims=1)
      GET = return %_AX.a_max[$[1]];
    MA_MAX_AX_VELO $MA_MAX_AX_VELO (ArrayDims=1)
      GET = return %_AX.v_max[$[1]];
    MA_MAX_AX_JERK $MA_MAX_AX_JERK (ArrayDims=1)
      GET = return %_AX.jerk_max[$[1]];
    MA_POSCTRL_GAIN $MA_POSCTRL_GAIN (ArrayDims=1)
      GET = return %_AX.servo_gain[$[1]];
    MA_REFP_SET_POS $MA_REFP_SET_POS (ArrayDims=1)
      GET = return %_AX.home_pos[$[1]];
    MA_POS_LIMIT_PLUS $MA_POS_LIMIT_PLUS (ArrayDims=1)
      GET = return %_AX.pos_sw_end[$[1]];
    MA_POS_LIMIT_MINUS $MA_POS_LIMIT_MINUS (ArrayDims=1)
      GET = return %_AX.neg_sw_end[$[1]];
  Parameters:
    R (IndexType=RParamIndex, ValueType=FLOAT)
      ARG (ref=EXPR, DataType=RParamIndex)
    QUOTED (QuotedName=$R, Synchronous=Yes, IndexType=RParamIndex, ValueType=FLOAT)
      ARG (ref=EXPR, DataType=RParamIndex)
    QUOTED (QuotedName=$P, Synchronous=Yes, IndexType=RParamIndex, ValueType=FLOAT)
      ARG (ref=EXPR, DataType=RParamIndex)
    EXB (IndexType=EXParamIndex, ValueType=Byte)
      ARG (ref=EXPR, DataType=EXParamIndex)
    EXW (IndexType=EXParamIndex, ValueType=Word)
      ARG (ref=EXPR, DataType=EXParamIndex)
    EXL (IndexType=EXParamIndex, ValueType=Long)
      ARG (ref=EXPR, DataType=EXParamIndex)
    EXF (IndexType=EXFParamIndex, ValueType=FLOAT)
      ARG (ref=EXPR, DataType=EXFParamIndex)
    MW (Synchronous=Yes, IndexType=MParamIndex, ValueType=Word)
      ARG (ref=EXPR, DataType=MParamIndex)
    ML (Synchronous=Yes, IndexType=MParamIndex, ValueType=Long)
      ARG (ref=EXPR, DataType=MParamIndex)
    MF (Synchronous=Yes, IndexType=MParamIndex, ValueType=FLOAT)
      ARG (ref=EXPR, DataType=MParamIndex)
  MCodes:
    M17 = 17 (Group=41, Alias=RET:[^\d\w\(], Eval=Early, Inline=Yes, AliasIsPattern=Yes)
      ARG (ref=VALUE, DataType=FLOAT, RequireLiteral=Yes)
    M17_1 = 17.1 (Group=41, Alias=CONDRET, Eval=Early, Inline=Yes)
      ARG (ref=VALUE, DataType=FLOAT, RequireLiteral=Yes)
```

- Data object Logical/GmcIpConfig/gmcipesm (Cnc, version 2.48.1) (no source held here)
